// TIA Portal project "2022.05.03_红绿灯" (V17)

(* hardware
DEVICE "S7-1500/ET200MP station_1"  S7-1500 station
   slot 0: "导轨_0"  Rack  6ES7 590-1***0-0AA0
   slot 1: "PLC_1"  CPU 1516-3 PN/DP  6ES7 516-3AN00-0AB0  V1.7
      slot 3: "CPU 显示_1"  6ES7591-1BA00-0AA0
      slot 32768: "PROFINET 接口_1"  X1
         slot 32769: "端口_1"  X1 P1
         slot 32770: "端口_2"  X1 P2
      slot 33024: "PROFINET 接口_2"  X2
         slot 33025: "端口_1"  X2 P1
      slot 33280: "DP 接口_1"  X3
   slot 2: "DI 32x24VDC BA_1"  DI 32x24VDC BA  6ES7 521-1BL10-0AA0  V1.1
   slot 3: "DQ 32x24VDC/0.5A HF_1"  DQ 32x24VDC/0.5A HF  6ES7 522-1BL01-0AB0  V1.1
*)

// ===== PLC "PLC_1"  CPU 1516-3 PN/DP =====

VAR_GLOBAL   // PLC tag table "默认变量表"
   "按钮1" AT %I0.0 : Bool;
   "按钮2" AT %I0.1 : Bool;
   "按钮3" AT %I0.2 : Bool;
   "按钮4" AT %I0.3 : Bool;
   "按钮5" AT %I0.4 : Bool;
   "按钮6" AT %I0.5 : Bool;
   "按钮7" AT %I0.6 : Bool;
   "按钮8" AT %I0.7 : Bool;
   "按钮9" AT %I1.0 : Bool;
   "按钮10" AT %I1.1 : Bool;
   "按钮11" AT %I1.2 : Bool;
   "指示灯1" AT %Q0.0 : Bool;
   "指示灯2" AT %Q0.1 : Bool;
   "指示灯3" AT %Q0.2 : Bool;
   "指示灯4" AT %Q0.3 : Bool;
   "指示灯5" AT %Q0.4 : Bool;
   "指示灯6" AT %Q0.5 : Bool;
   "指示灯7" AT %Q0.6 : Bool;
   "指示灯8" AT %Q0.7 : Bool;
   "指示灯9" AT %Q1.0 : Bool;
   "指示灯10" AT %Q1.1 : Bool;
   "指示灯11" AT %Q1.2 : Bool;
   "指示灯12" AT %Q1.3 : Bool;
   "北红灯" AT %M20.0 : Bool;
   "北绿灯" AT %M20.1 : Bool;
   "北黄灯" AT %M20.2 : Bool;
   "南红灯" AT %M20.3 : Bool;
   "南绿灯" AT %M20.4 : Bool;
   "南黄灯" AT %M20.5 : Bool;
   "西红灯" AT %M20.6 : Bool;
   "西绿灯" AT %M20.7 : Bool;
   "西黄灯" AT %M21.0 : Bool;
   "东红灯" AT %M21.1 : Bool;
   "东绿灯" AT %M21.2 : Bool;
   "东黄灯" AT %M21.3 : Bool;
   "测试" AT %M50.0 : Bool;
   "设备启动" AT %M50.1 : Bool;
   "设备停止" AT %M50.2 : Bool;
   "Clock_Byte(1)" AT %MB0 : Byte;
   "Clock_10Hz(1)" AT %M0.0 : Bool;
   "Clock_5Hz" AT %M0.1 : Bool;
   "Clock_2.5Hz" AT %M0.2 : Bool;
   "Clock_2Hz" AT %M0.3 : Bool;
   "Clock_1.25Hz" AT %M0.4 : Bool;
   "Clock_1Hz" AT %M0.5 : Bool;
   "Clock_0.625Hz" AT %M0.6 : Bool;
   "Clock_0.5Hz" AT %M0.7 : Bool;
   "启动" AT %M50.3 : Bool;
   "南北黄灯保持" AT %M50.5 : Bool;
   "东西黄灯保持" AT %M50.6 : Bool;
   "1" AT %M1.0 : Bool;
   "0" AT %M1.1 : Bool;
END_VAR

DATA_BLOCK "灯定时器"   // DB1
{ S7_Optimized_Access := 'TRUE' }
VERSION : 0.1
   VAR
      南北红灯 : IEC_TIMER;
      南北绿灯 : IEC_TIMER;
      南北黄灯 : IEC_TIMER;
      东西绿灯 : IEC_TIMER;
      东西红灯 : IEC_TIMER;
      东西黄灯 : IEC_TIMER;
      定时器Q : Struct
         南北红灯Q : Bool;
         南北绿灯Q : Bool;
         南北黄灯Q : Bool;
         东西绿灯Q : Bool;
         东西红灯Q : Bool;
         东西黄灯Q : Bool;
      END_STRUCT;
   END_VAR
BEGIN
END_DATA_BLOCK

FUNCTION "计数器控制LAD" : Void   // FC1, LAD
{ S7_Optimized_Access := 'TRUE' }
VERSION : 0.1
   VAR_TEMP   // added for the SCL form of the ladder/FBD networks
      _w1 : Bool;
   END_VAR
BEGIN

REGION Network 1: 启动停止程序
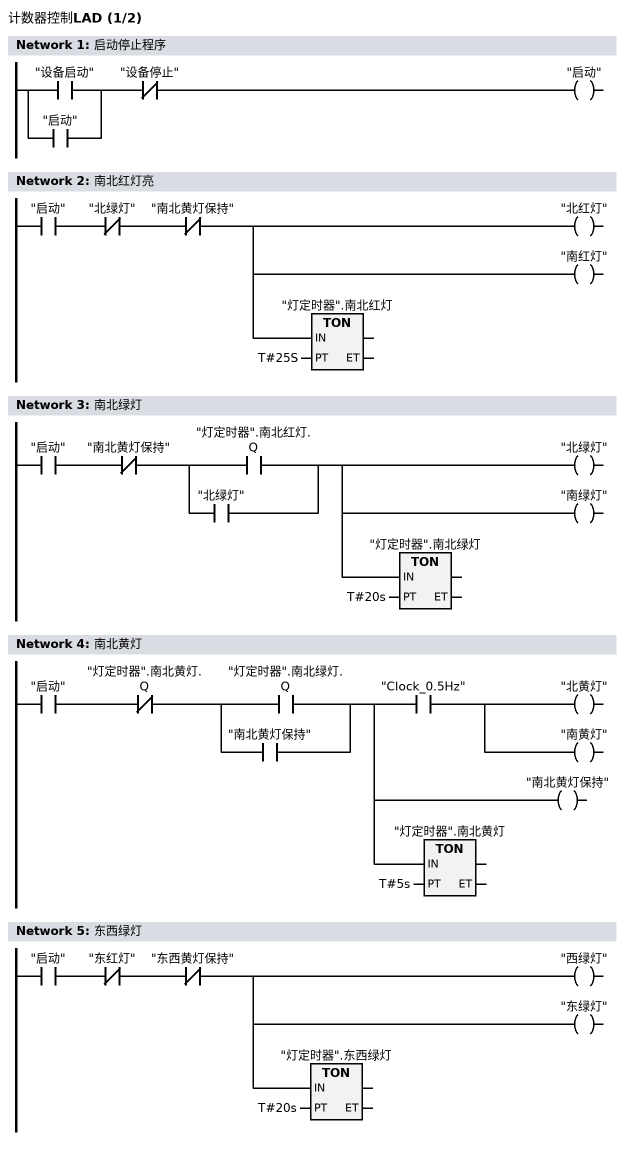
   RUNG wire#powerrail
      Contact( "设备启动" )
      wire#w1
      I_Contact( "设备停止" )
      Coil( "启动" )
   END_RUNG
   RUNG wire#powerrail
      Contact( "启动" )
   END_RUNG wire#w1
   // the same network as SCL:
   "启动" := ("设备启动" OR "启动") AND NOT "设备停止";
END_REGION

REGION Network 2: 南北红灯亮
   "北红灯" := "启动" AND NOT "北绿灯" AND NOT "南北黄灯保持";
   "南红灯" := "北红灯";
   "灯定时器".南北红灯.TON(IN := "北红灯", PT := T#25S);
END_REGION

REGION Network 3: 南北绿灯
   "北绿灯" := "启动" AND NOT "南北黄灯保持" AND ("灯定时器".南北红灯.Q OR "北绿灯");
   "南绿灯" := "北绿灯";
   "灯定时器".南北绿灯.TON(IN := "北绿灯", PT := T#20s);
END_REGION

REGION Network 4: 南北黄灯
   #_w1 := "启动" AND NOT "灯定时器".南北黄灯.Q AND ("灯定时器".南北绿灯.Q OR "南北黄灯保持");
   "北黄灯" := #_w1 AND "Clock_0.5Hz";
   "南黄灯" := "北黄灯";
   "南北黄灯保持" := #_w1;
   "灯定时器".南北黄灯.TON(IN := #_w1, PT := T#5s);
END_REGION

REGION Network 5: 东西绿灯
   "西绿灯" := "启动" AND NOT "东红灯" AND NOT "东西黄灯保持";
   "东绿灯" := "西绿灯";
   "灯定时器".东西绿灯.TON(IN := "西绿灯", PT := T#20s);
END_REGION

REGION Network 6: 东西黄灯
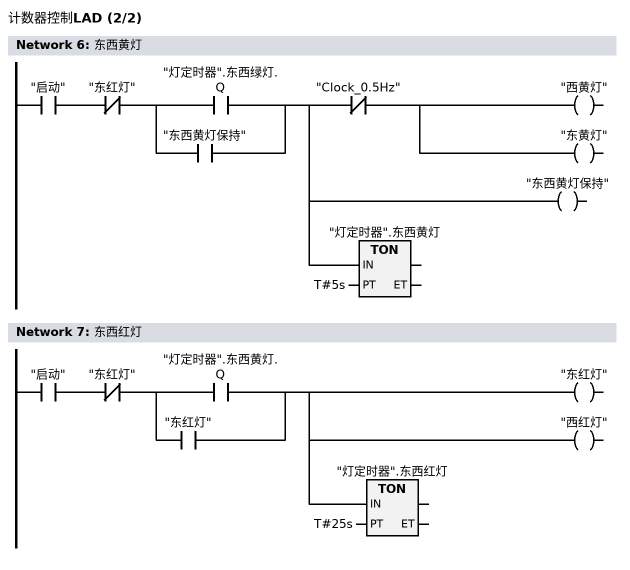
   #_w1 := "启动" AND NOT "东红灯" AND ("灯定时器".东西绿灯.Q OR "东西黄灯保持");
   "西黄灯" := #_w1 AND NOT "Clock_0.5Hz";
   "东黄灯" := "西黄灯";
   "东西黄灯保持" := #_w1;
   "灯定时器".东西黄灯.TON(IN := #_w1, PT := T#5s);
END_REGION

REGION Network 7: 东西红灯
   "东红灯" := "启动" AND NOT "东红灯" AND ("灯定时器".东西黄灯.Q OR "东红灯");
   "西红灯" := "东红灯";
   "灯定时器".东西红灯.TON(IN := "东红灯", PT := T#25s);
END_REGION
END_FUNCTION

FUNCTION "红绿灯FBD" : Void   // FC2, FBD
{ S7_Optimized_Access := 'TRUE' }
VERSION : 0.1
   VAR_TEMP   // added for the SCL form of the ladder/FBD networks
      _w1 : Bool;
   END_VAR
BEGIN

REGION Network 1: 启动停止程序
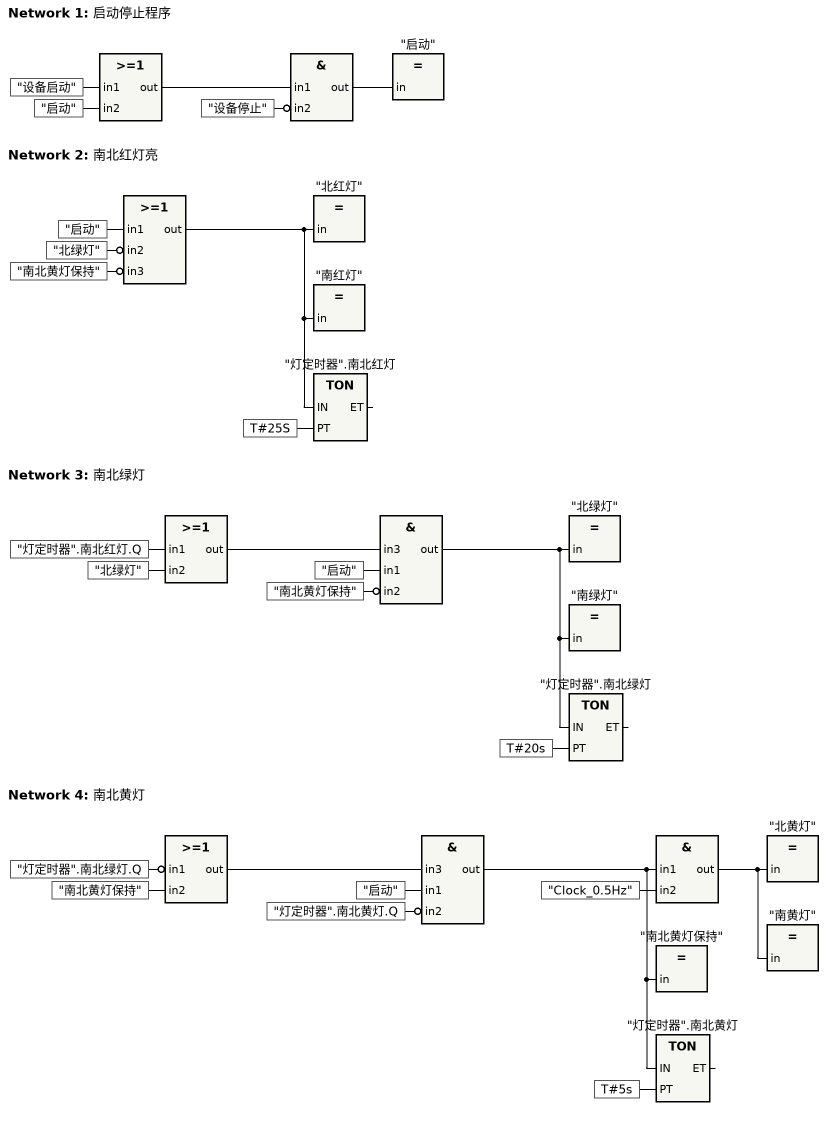
   "启动" := ("设备启动" OR "启动") AND NOT "设备停止";
END_REGION

REGION Network 2: 南北红灯亮
   "北红灯" := "启动" OR NOT "北绿灯" OR NOT "南北黄灯保持";
   "南红灯" := "北红灯";
   "灯定时器".南北红灯.TON(IN := "北红灯", PT := T#25S);
END_REGION

REGION Network 3: 南北绿灯
   "北绿灯" := ("灯定时器".南北红灯.Q OR "北绿灯") AND "启动" AND NOT "南北黄灯保持";
   "南绿灯" := "北绿灯";
   "灯定时器".南北绿灯.TON(IN := "北绿灯", PT := T#20s);
END_REGION

REGION Network 4: 南北黄灯
   #_w1 := (NOT "灯定时器".南北绿灯.Q OR "南北黄灯保持") AND "启动" AND NOT "灯定时器".南北黄灯.Q;
   "北黄灯" := #_w1 AND "Clock_0.5Hz";
   "南黄灯" := "北黄灯";
   "南北黄灯保持" := #_w1;
   "灯定时器".南北黄灯.TON(IN := #_w1, PT := T#5s);
END_REGION

REGION Network 5: 东西绿灯
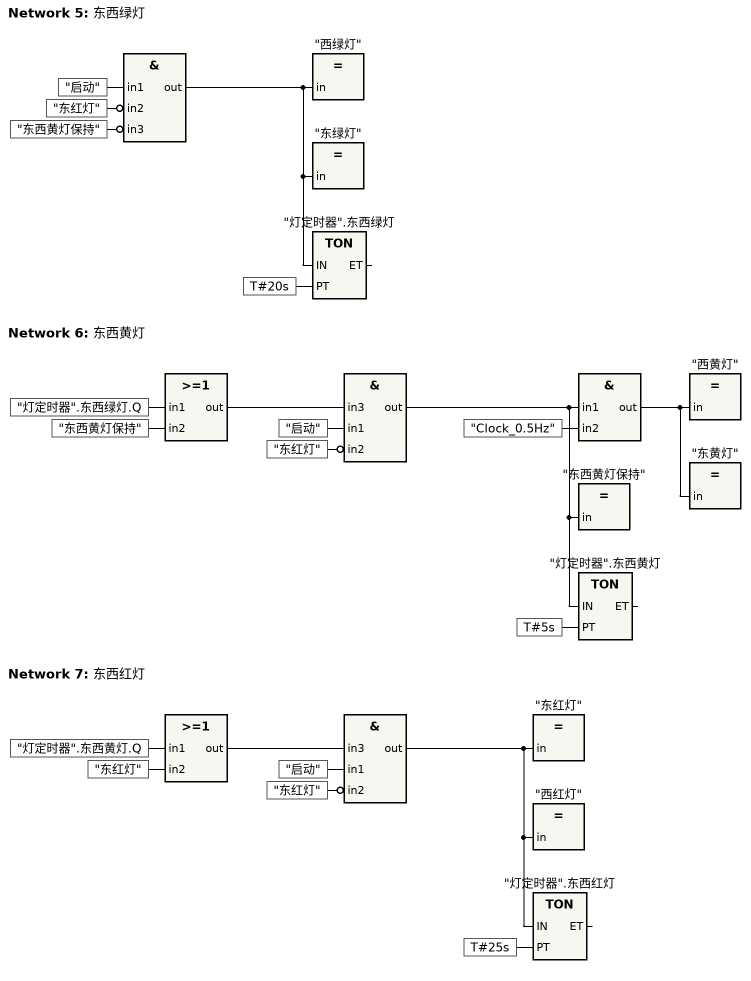
   "西绿灯" := "启动" AND NOT "东红灯" AND NOT "东西黄灯保持";
   "东绿灯" := "西绿灯";
   "灯定时器".东西绿灯.TON(IN := "西绿灯", PT := T#20s);
END_REGION

REGION Network 6: 东西黄灯
   #_w1 := ("灯定时器".东西绿灯.Q OR "东西黄灯保持") AND "启动" AND NOT "东红灯";
   "西黄灯" := #_w1 AND "Clock_0.5Hz";
   "东黄灯" := "西黄灯";
   "东西黄灯保持" := #_w1;
   "灯定时器".东西黄灯.TON(IN := #_w1, PT := T#5s);
END_REGION

REGION Network 7: 东西红灯
   "东红灯" := ("灯定时器".东西黄灯.Q OR "东红灯") AND "启动" AND NOT "东红灯";
   "西红灯" := "东红灯";
   "灯定时器".东西红灯.TON(IN := "东红灯", PT := T#25s);
END_REGION
END_FUNCTION

FUNCTION "红绿灯控制SCL" : Void   // FC3, SCL
{ S7_Optimized_Access := 'TRUE' }
VERSION : 0.1
BEGIN
   //启动停止程序
   IF "设备启动" OR "启动" THEN
       IF "设备停止" = 0 THEN
           "启动" := 1;
       ELSE
           "启动" := 0;
       END_IF;
   END_IF;

   //南北红灯亮
   IF "启动" AND "北绿灯" = 0 AND "南北黄灯保持" = 0 THEN
       "北红灯" := 1;
       "南红灯" := 1;
       "灯定时器".南北红灯.TON(IN := "北红灯",
                       PT := T#25S,
                       Q => "灯定时器".定时器Q.南北红灯Q
       );
   ELSE
       "北红灯" := 0;
       "南红灯" := 0;
       RESET_TIMER("灯定时器".南北红灯);
       "灯定时器".定时器Q.南北红灯Q := 0;
   END_IF;

   //南北绿灯
   IF "启动" AND "南北黄灯保持"=0 THEN
       IF "灯定时器".定时器Q.南北绿灯Q OR "北绿灯" THEN
           "北绿灯" := 1;
           "南绿灯" := 1;
           "灯定时器".南北绿灯.TON(IN := "北绿灯",
                           PT := T#20S,
                           Q => "灯定时器".定时器Q.南北绿灯Q);
       ELSE
           "北绿灯" := 0;
           "南绿灯" := 0;
           RESET_TIMER("灯定时器".南北绿灯);
           "灯定时器".定时器Q.南北绿灯Q := 0;
       END_IF;
   ELSE
       "北绿灯" := 0;
       "南绿灯" := 0;
       RESET_TIMER("灯定时器".南北绿灯);
       "灯定时器".定时器Q.南北绿灯Q := 0;
   END_IF;

   //南北黄灯
   IF "启动" AND "灯定时器".定时器Q.南北黄灯Q = 0 THEN
       IF "灯定时器".定时器Q.南北绿灯Q OR "南北黄灯保持" THEN
           IF "Clock_0.5Hz" THEN
               "北黄灯" := 1;
               "南黄灯" := 1;
           ELSE
               "北黄灯" := 0;
               "南黄灯" := 0;
           END_IF;
           "南北黄灯保持" := 1;
           "灯定时器".南北黄灯.TON(IN := "南北黄灯保持",
                           PT := T#5S,
                           Q => "灯定时器".定时器Q.南北黄灯Q);
       ELSE
           "北黄灯" := 0;
           "南黄灯" := 0;
           "灯定时器".定时器Q.南北黄灯Q := 0;
           RESET_TIMER("灯定时器".南北黄灯);
       END_IF;
   ELSE
       "北黄灯" := 0;
       "南黄灯" := 0;
       "灯定时器".定时器Q.南北黄灯Q := 0;
       RESET_TIMER("灯定时器".南北黄灯);
   END_IF;

   //东西绿灯
   IF "启动" AND "东红灯" = 0 AND "东西黄灯保持" = 0 THEN
       "西绿灯" := 1;
       "东绿灯" := 1;
       "灯定时器".南北绿灯.TON(IN := "西绿灯",
                       PT := T#20S,
                       Q => "灯定时器".定时器Q.南北绿灯Q);
   ELSE
       "西绿灯" := 0;
       "东绿灯" := 0;
       RESET_TIMER("灯定时器".南北绿灯);
       "灯定时器".定时器Q.南北绿灯Q := 0;
   END_IF;

    //东西黄灯
   IF "启动" AND "东红灯" = 0 THEN
       IF "灯定时器".东西绿灯.Q OR "东西黄灯保持" THEN
           IF "Clock_0.5Hz" THEN
               "西黄灯" := 1;
               "东黄灯" := 1;
           ELSE
               "西黄灯" := 0;
               "东黄灯" := 0;
           END_IF;
           "东西黄灯保持" := 1;
           "灯定时器".东西黄灯.TON(IN := "东西黄灯保持",
                           PT := T#5S,
                           Q => "灯定时器".定时器Q.东西黄灯Q);
       ELSE
           "西黄灯" := 0;
           "东黄灯" := 0;
           "东西黄灯保持" := "0";
           RESET_TIMER("灯定时器".东西黄灯);
           "灯定时器".定时器Q.东西黄灯Q := 0;
       END_IF;
   ELSE
       "西黄灯" := 0;
       "东黄灯" := 0;
       "东西黄灯保持" := "0";
       RESET_TIMER("灯定时器".东西黄灯);
       "灯定时器".定时器Q.东西黄灯Q := 0;
   END_IF;

   //东西红灯
   IF "启动" AND "东红灯"=0 THEN
       IF "灯定时器".东西黄灯.Q AND "东红灯" THEN
           "东红灯" := 1;
           "西红灯" := 1;
           "灯定时器".东西红灯.TON(IN := "东红灯",
                           PT := T#25S,
                           Q => "灯定时器".定时器Q.东西红灯Q);
       ELSE
           "东红灯" := 0;
           "西红灯" := 0;
           RESET_TIMER("灯定时器".东西红灯);
           "灯定时器".定时器Q.东西红灯Q := 0;
       END_IF;
   ELSE
       "东红灯" := 0;
       "西红灯" := 0;
       RESET_TIMER("灯定时器".东西红灯);
       "灯定时器".定时器Q.东西红灯Q := 0;
   END_IF;
END_FUNCTION

ORGANIZATION_BLOCK "Main"   // OB1, LAD, ProgramCycle
TITLE = "Main Program Sweep (Cycle)"
{ S7_Optimized_Access := 'TRUE' }
VERSION : 0.1
   VAR_INPUT
      Initial_Call : Bool;   // Initial call of this OB
      Remanence : Bool;   // =True, if remanent data are available
   END_VAR
BEGIN

REGION Network 1
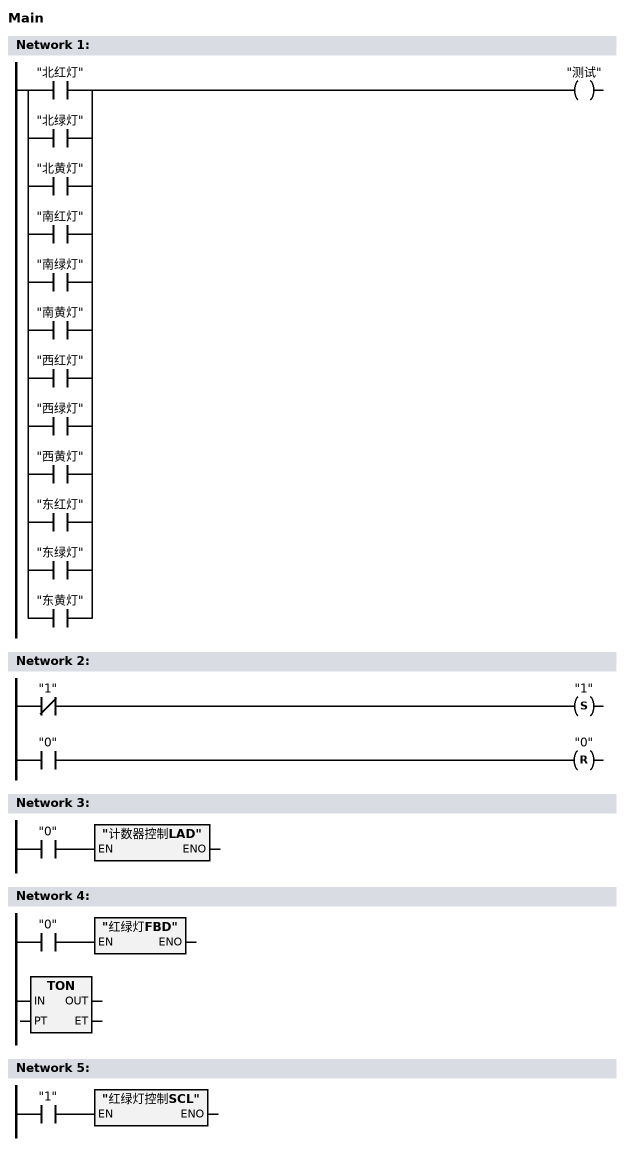
   RUNG wire#powerrail
      Contact( "北红灯" )
      wire#w1
      Coil( "测试" )
   END_RUNG
   RUNG wire#powerrail
      Contact( "北绿灯" )
   END_RUNG wire#w1
   RUNG wire#powerrail
      Contact( "北黄灯" )
   END_RUNG wire#w1
   RUNG wire#powerrail
      Contact( "南红灯" )
   END_RUNG wire#w1
   RUNG wire#powerrail
      Contact( "南绿灯" )
   END_RUNG wire#w1
   RUNG wire#powerrail
      Contact( "南黄灯" )
   END_RUNG wire#w1
   RUNG wire#powerrail
      Contact( "西红灯" )
   END_RUNG wire#w1
   RUNG wire#powerrail
      Contact( "西绿灯" )
   END_RUNG wire#w1
   RUNG wire#powerrail
      Contact( "西黄灯" )
   END_RUNG wire#w1
   RUNG wire#powerrail
      Contact( "东红灯" )
   END_RUNG wire#w1
   RUNG wire#powerrail
      Contact( "东绿灯" )
   END_RUNG wire#w1
   RUNG wire#powerrail
      Contact( "东黄灯" )
   END_RUNG wire#w1
   // the same network as SCL:
   "测试" := "北红灯" OR "北绿灯" OR "北黄灯" OR "南红灯" OR "南绿灯" OR "南黄灯" OR "西红灯" OR "西绿灯" OR "西黄灯" OR "东红灯" OR "东绿灯" OR "东黄灯";
END_REGION

REGION Network 2
   RUNG wire#powerrail
      I_Contact( "1" )
      S_Coil( "1" )
   END_RUNG
   RUNG wire#powerrail
      Contact( "0" )
      R_Coil( "0" )
   END_RUNG
   // the same network as SCL:
   IF NOT "1" THEN "1" := TRUE; END_IF;
   IF "0" THEN "0" := FALSE; END_IF;
END_REGION

REGION Network 3
   RUNG wire#powerrail
      Contact( "0" )
      "计数器控制LAD"()
   END_RUNG
   // the same network as SCL:
   IF "0" THEN "计数器控制LAD"(); END_IF;
END_REGION

REGION Network 4
   IF "0" THEN "红绿灯FBD"(); END_IF;
   TON(IN := TRUE);
END_REGION

REGION Network 5
   RUNG wire#powerrail
      Contact( "1" )
      "红绿灯控制SCL"()
   END_RUNG
   // the same network as SCL:
   IF "1" THEN "红绿灯控制SCL"(); END_IF;
END_REGION
END_ORGANIZATION_BLOCK